{attribute 'qualified_only'}
{attribute 'strict'}
TYPE E_Compare :
(
	EQUAL,
	NOT_EQUAL,
	LESS_THAN,
	LOWER_THAN_OR_EQUAL,
	GREATER_THAN,
	GREATER_THAN_OR_EQUAL
);
END_TYPE

(* stored: Version 1.1.0.1, ProductVersion 3.1.4024.11
   DUT E_Compare: Id {102e080b-da02-4c0b-a370-e824c6e3fd0b} *)
